FUNCTION DriveOperatingModesToString : STRING
VAR_INPUT
    mode : DriveOperatingModes;
END_VAR
VAR
END_VAR

CASE mode OF
    
    DriveOperatingModes.OPERATING_MODE_NONE:
        DriveOperatingModesToString := 'None';
    DriveOperatingModes.OPERATING_MODE_TORQUE_CONTROL:
        DriveOperatingModesToString := 'Torque control';
    DriveOperatingModes.OPERATING_MODE_VELOCITY_CONTROL:
        DriveOperatingModesToString := 'Velocity control';
    DriveOperatingModes.OPERATING_MODE_POSITION_CONTROL:
        DriveOperatingModesToString := 'Position control';

END_CASE

END_FUNCTION

(* stored: Version 1.1.0.1, ProductVersion 3.1.4018.5
   POU DriveOperatingModesToString: Id {4fc7bd17-6ec2-43ad-b516-f822d5b5ec0a}, SpecialFunc None *)
